// LS Electric XG5000 project: 8_26
// PLC LSPLC
// module base 0 slot 0: 입출력 모듈:XBC-DR14E (DC 24V 입력 8점, 릴레이 출력 6점)

PROGRAM NewProgram (task: 스캔 프로그램)

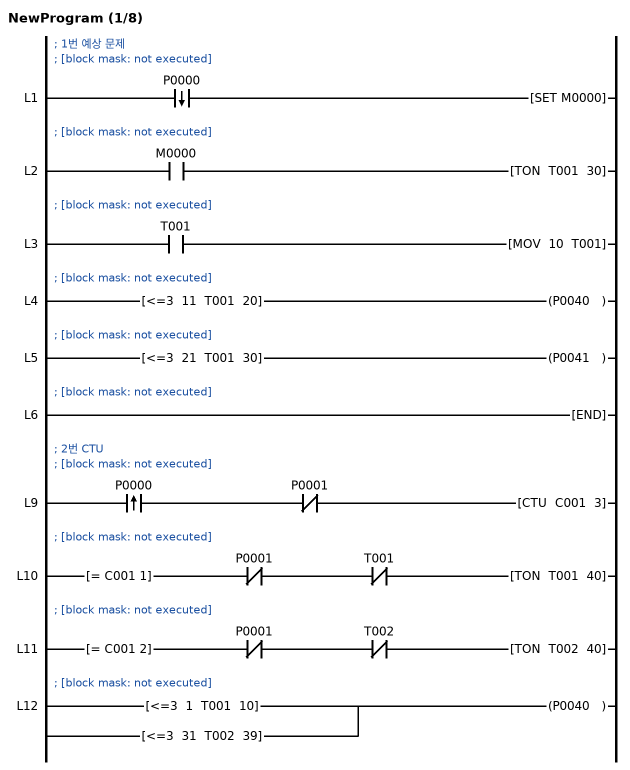
// 1번 예상 문제
; L1 (block mask: not executed)
LOADN     P0000
SET       M0000
; L2 (block mask: not executed)
LOAD      M0000
TON       T001 30
; L3 (block mask: not executed)
LOAD      T001
MOV       10 T001
; L4 (block mask: not executed)
LOAD<=3   11 T001 20
OUT       P0040
; L5 (block mask: not executed)
LOAD<=3   21 T001 30
OUT       P0041
; L6 (block mask: not executed)
END
// 2번 CTU
; L9 (block mask: not executed)
LOADP     P0000
AND NOT   P0001
CTU       C001 3
; L10 (block mask: not executed)
LOAD=     C001 1
AND NOT   P0001
AND NOT   T001
TON       T001 40
; L11 (block mask: not executed)
LOAD=     C001 2
AND NOT   P0001
AND NOT   T002
TON       T002 40
; L12 (block mask: not executed)
LOAD<=3   1 T001 10
OR<=3     31 T002 39
OUT       P0040

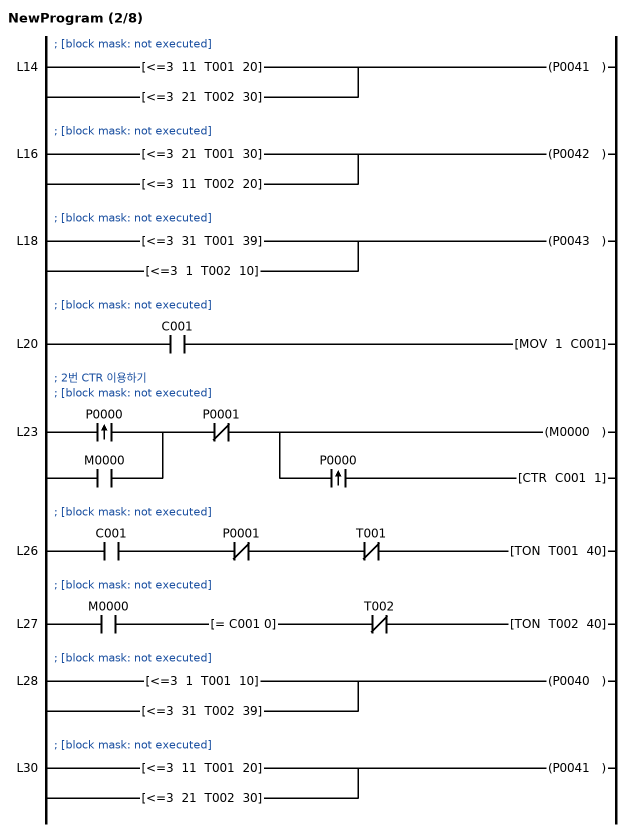
; L14 (block mask: not executed)
LOAD<=3   11 T001 20
OR<=3     21 T002 30
OUT       P0041
; L16 (block mask: not executed)
LOAD<=3   21 T001 30
OR<=3     11 T002 20
OUT       P0042
; L18 (block mask: not executed)
LOAD<=3   31 T001 39
OR<=3     1 T002 10
OUT       P0043
; L20 (block mask: not executed)
LOAD      C001
MOV       1 C001
// 2번 CTR 이용하기
; L23 (block mask: not executed)
LOADP     P0000
OR        M0000
AND NOT   P0001
OUT       M0000
ANDP      P0000
CTR       C001 1
; L26 (block mask: not executed)
LOAD      C001
AND NOT   P0001
AND NOT   T001
TON       T001 40
; L27 (block mask: not executed)
LOAD      M0000
AND=      C001 0
AND NOT   T002
TON       T002 40
; L28 (block mask: not executed)
LOAD<=3   1 T001 10
OR<=3     31 T002 39
OUT       P0040
; L30 (block mask: not executed)
LOAD<=3   11 T001 20
OR<=3     21 T002 30
OUT       P0041

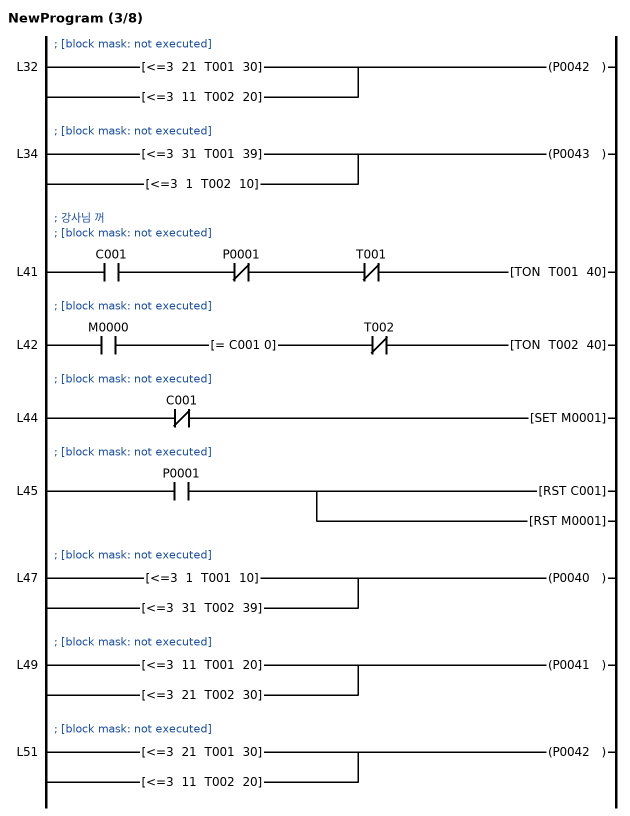
; L32 (block mask: not executed)
LOAD<=3   21 T001 30
OR<=3     11 T002 20
OUT       P0042
; L34 (block mask: not executed)
LOAD<=3   31 T001 39
OR<=3     1 T002 10
OUT       P0043
// 강사님 꺼
; L41 (block mask: not executed)
LOAD      C001
AND NOT   P0001
AND NOT   T001
TON       T001 40
; L42 (block mask: not executed)
LOAD      M0000
AND=      C001 0
AND NOT   T002
TON       T002 40
; L44 (block mask: not executed)
LOAD NOT  C001
SET       M0001
; L45 (block mask: not executed)
LOAD      P0001
RST       C001
RST       M0001
; L47 (block mask: not executed)
LOAD<=3   1 T001 10
OR<=3     31 T002 39
OUT       P0040
; L49 (block mask: not executed)
LOAD<=3   11 T001 20
OR<=3     21 T002 30
OUT       P0041
; L51 (block mask: not executed)
LOAD<=3   21 T001 30
OR<=3     11 T002 20
OUT       P0042

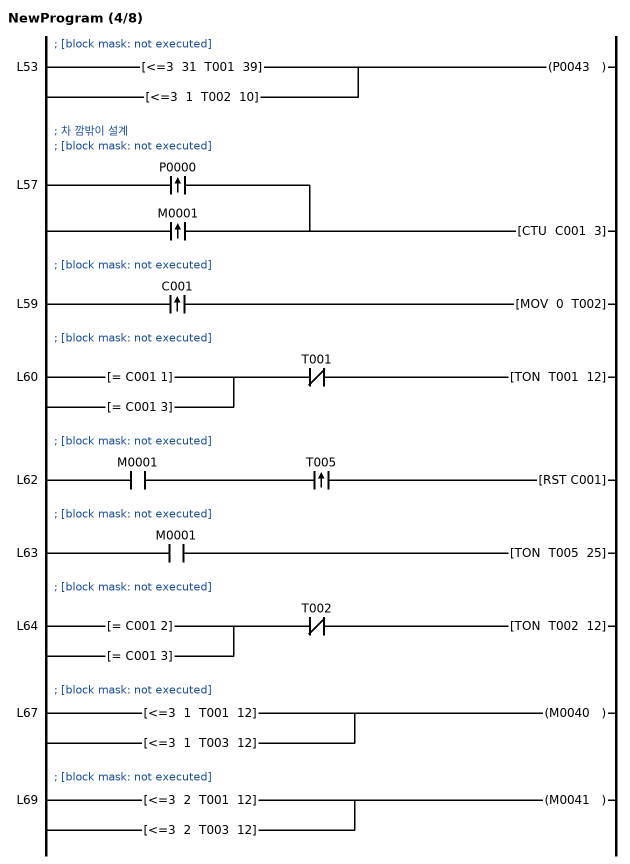
; L53 (block mask: not executed)
LOAD<=3   31 T001 39
OR<=3     1 T002 10
OUT       P0043
// 차 깜밖이 설계
; L57 (block mask: not executed)
LOADP     P0000
ORP       M0001
CTU       C001 3
; L59 (block mask: not executed)
LOADP     C001
MOV       0 T002
; L60 (block mask: not executed)
LOAD=     C001 1
OR=       C001 3
AND NOT   T001
TON       T001 12
; L62 (block mask: not executed)
LOAD      M0001
ANDP      T005
RST       C001
; L63 (block mask: not executed)
LOAD      M0001
TON       T005 25
; L64 (block mask: not executed)
LOAD=     C001 2
OR=       C001 3
AND NOT   T002
TON       T002 12
; L67 (block mask: not executed)
LOAD<=3   1 T001 12
OR<=3     1 T003 12
OUT       M0040
; L69 (block mask: not executed)
LOAD<=3   2 T001 12
OR<=3     2 T003 12
OUT       M0041

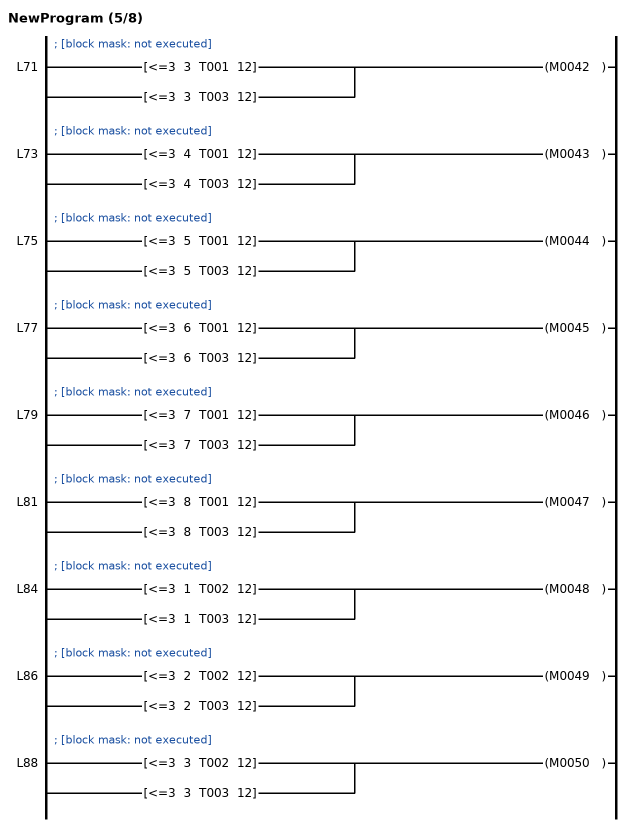
; L71 (block mask: not executed)
LOAD<=3   3 T001 12
OR<=3     3 T003 12
OUT       M0042
; L73 (block mask: not executed)
LOAD<=3   4 T001 12
OR<=3     4 T003 12
OUT       M0043
; L75 (block mask: not executed)
LOAD<=3   5 T001 12
OR<=3     5 T003 12
OUT       M0044
; L77 (block mask: not executed)
LOAD<=3   6 T001 12
OR<=3     6 T003 12
OUT       M0045
; L79 (block mask: not executed)
LOAD<=3   7 T001 12
OR<=3     7 T003 12
OUT       M0046
; L81 (block mask: not executed)
LOAD<=3   8 T001 12
OR<=3     8 T003 12
OUT       M0047
; L84 (block mask: not executed)
LOAD<=3   1 T002 12
OR<=3     1 T003 12
OUT       M0048
; L86 (block mask: not executed)
LOAD<=3   2 T002 12
OR<=3     2 T003 12
OUT       M0049
; L88 (block mask: not executed)
LOAD<=3   3 T002 12
OR<=3     3 T003 12
OUT       M0050

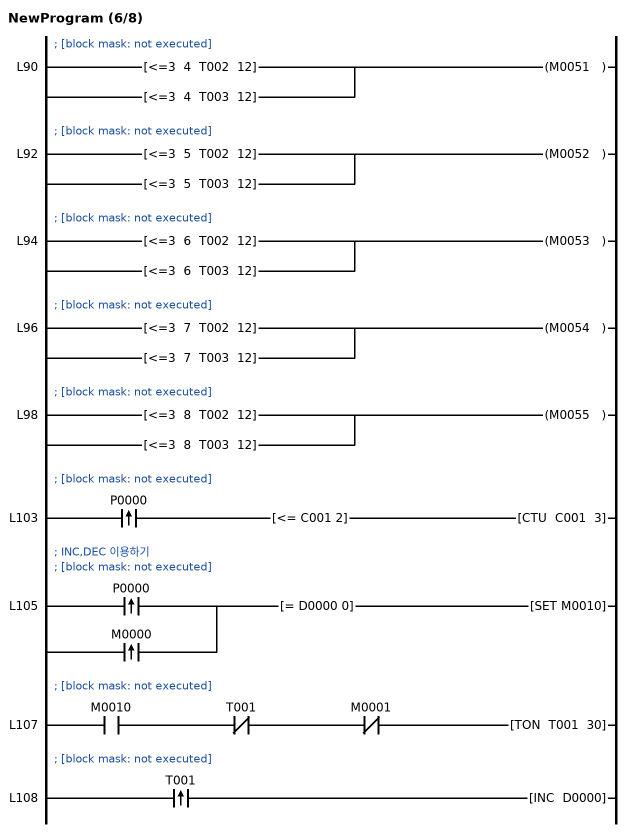
; L90 (block mask: not executed)
LOAD<=3   4 T002 12
OR<=3     4 T003 12
OUT       M0051
; L92 (block mask: not executed)
LOAD<=3   5 T002 12
OR<=3     5 T003 12
OUT       M0052
; L94 (block mask: not executed)
LOAD<=3   6 T002 12
OR<=3     6 T003 12
OUT       M0053
; L96 (block mask: not executed)
LOAD<=3   7 T002 12
OR<=3     7 T003 12
OUT       M0054
; L98 (block mask: not executed)
LOAD<=3   8 T002 12
OR<=3     8 T003 12
OUT       M0055
; L103 (block mask: not executed)
LOADP     P0000
AND<=     C001 2
CTU       C001 3
// INC,DEC 이용하기
; L105 (block mask: not executed)
LOADP     P0000
ORP       M0000
AND=      D0000 0
SET       M0010
; L107 (block mask: not executed)
LOAD      M0010
AND NOT   T001
AND NOT   M0001
TON       T001 30
; L108 (block mask: not executed)
LOADP     T001
INC       D0000

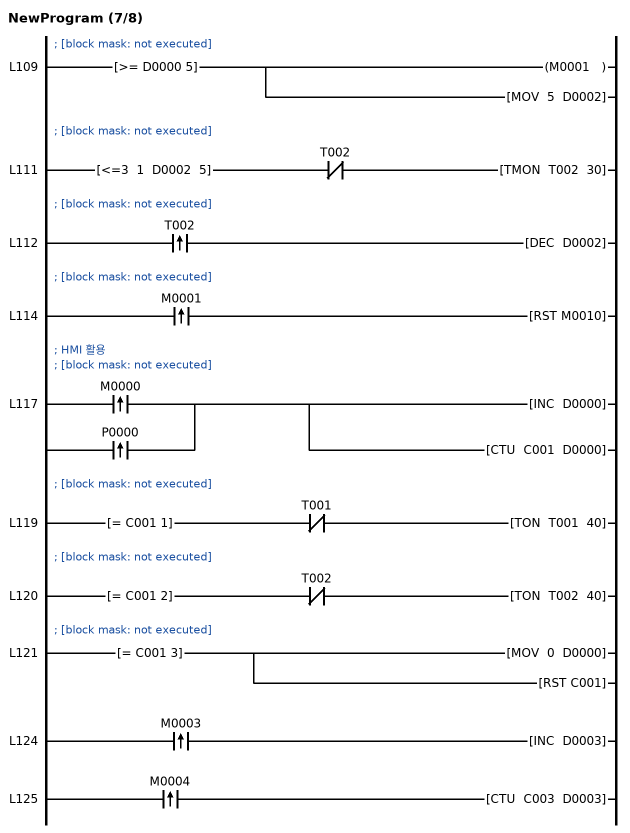
; L109 (block mask: not executed)
LOAD>=    D0000 5
OUT       M0001
MOV       5 D0002
; L111 (block mask: not executed)
LOAD<=3   1 D0002 5
AND NOT   T002
TMON      T002 30
; L112 (block mask: not executed)
LOADP     T002
DEC       D0002
; L114 (block mask: not executed)
LOADP     M0001
RST       M0010
// HMI 활용
; L117 (block mask: not executed)
LOADP     M0000
ORP       P0000
INC       D0000
CTU       C001 D0000
; L119 (block mask: not executed)
LOAD=     C001 1
AND NOT   T001
TON       T001 40
; L120 (block mask: not executed)
LOAD=     C001 2
AND NOT   T002
TON       T002 40
; L121 (block mask: not executed)
LOAD=     C001 3
MOV       0 D0000
RST       C001
; L124
LOADP     M0003
INC       D0003
; L125
LOADP     M0004
CTU       C003 D0003

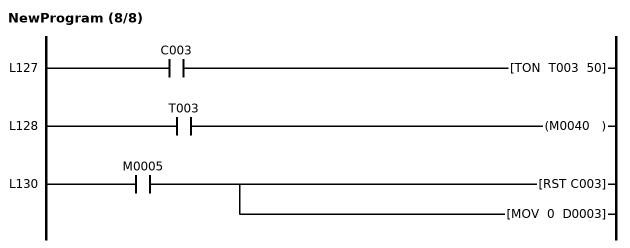
; L127
LOAD      C003
TON       T003 50
; L128
LOAD      T003
OUT       M0040
; L130
LOAD      M0005
RST       C003
MOV       0 D0003